{attribute addProperty BoxType "EQ3314-0002-0016"}
{attribute addProperty Id "TC_TCInputs_ChannelAT %I*ARRAY[0..3] OF TC_TCInputs_Channel_3FFCB36E128160WcStateAT %I*WcState_F855686C1620InfoDataAT %I*InfoData_BC63D37F80100"}
{attribute addProperty CRC "3647356279"}
{attribute addProperty SizeInBites "224"}
{attribute addProperty SizeInBytes "28"}
TYPE EQ3314_AF8E369F :
STRUCT
	{attribute addProperty Name "TC_TCInputs_Channel"}
	TC_TCInputs_Channel : ARRAY[0..3] OF TC_TCInputs_Channel_3FFCB36E;
	{attribute addProperty Name "WcState"}
	WcState : WcState_F855686C;
	{attribute addProperty Name "InfoData"}
	InfoData : InfoData_BC63D37F;
END_STRUCT
END_TYPE

(* stored: Version 1.2.0.0, ProductVersion 3.1.4024.9
   DUT EQ3314_AF8E369F: Id {f80c30b6-2f8c-4b93-b503-bd72268c7da4} *)
